FUNCTION_BLOCK ParserTestFbt1
END_FUNCTION_BLOCK
(* other elements stored in the file *)
(* pou name=functionBlock0 pouType=functionBlock *)
(* variable name=CTU0 *)
(* derived name=CTU *)
(* variable name=c *)
(* simpleValue value=false *)
(* block localId=1 typeName=CTU instanceName=CTU0 executionOrderId=0 *)
(* variable formalParameter=CU edge=rising *)
(* connection refLocalId=4 *)
(* variable formalParameter=R *)
(* connection refLocalId=6 *)
(* variable formalParameter=PV *)
(* variable formalParameter=Q *)
(* variable formalParameter=CV *)
(* outVariable localId=2 executionOrderId=0 negated=false *)
(* connection refLocalId=1 formalParameter=Q *)
(* expression  a *)
(* inOutVariable localId=3 executionOrderId=0 negatedOut=false negatedIn=false *)
(* connection refLocalId=1 formalParameter=CV *)
(* expression  b *)
(* inVariable localId=4 executionOrderId=0 negated=false *)
(* expression  c *)
(* continuation name=Connection0 localId=6 *)
